PROGRAM PRG_2_PMPS_PRE
VAR
END_VAR

MOTION_GVL.fbStandardPMPSDB(
    io_fbFFHWO:=GVL.fbFastFaultOutput1,
    bEnable:=TRUE,
    sPLCName:='kfe-motion',
);

END_PROGRAM

(* stored: Version 1.1.0.1, ProductVersion 3.1.4022.18
   POU PRG_2_PMPS_PRE: Id {3345ea47-dbca-467d-b104-e37cf5916a5b}, SpecialFunc None *)
